(* Logix 5000 project; controller test vendor 1 type 14 code 106 rev 30.11; software revision 30.00 *)

TASK MainTask (continuous, watchdog 500 ms) : MainProgram

MODULES
   Local : vendor 1 type 14 code 106 (Compact 0, rev 30.11)
END_MODULES

TYPE DateTime :   // Date and TimeOfDay (absolute) or Time (duration/interval)
STRUCT
   Yr : DINT;   // Year(s)
   Mo : DINT;   // Month(s)
   Da : DINT;   // Day(s)
   Hr : DINT;   // Hour(s)
   Min : DINT;   // Minute(s)
   Sec : DINT;   // Second(s)
   uSec : DINT;   // Microsecond(s)
END_STRUCT
END_TYPE

TYPE Diesel_User :
STRUCT
   user_number : DINT;   // user number/any 32 bit interger
   gallons_in : REAL;   // user gallons filled
   gallons_out : REAL;   // user gallons dispenced
   last_Tx : DateTime;   // date and time of last transaction
END_STRUCT
END_TYPE

ADD_ON_INSTRUCTION CALC_HORZ_TANK   (* revision 1.0, vendor truvision *)
// Gallons in a Horizontal Tank
// Help:
// Add on instruction to calculate the gallons in a cylindrical horizontal tank, based on the diameter of the tank, the length of the tank, and the distance from the surface of the liquid to the top of the tank.
VAR_INPUT
   cyl_dia : REAL; {required}
   cyl_len : REAL; {required}
   dist : REAL; {required}
END_VAR
VAR_IN_OUT
   gal : REAL; {required}
END_VAR
VAR
   al : REAL; {access None}
   vol : REAL; {access None}
   cyl_rad : REAL; {access None}
END_VAR

ROUTINE Logic   (* structured text *)
   cyl_rad:=cyl_dia/2;
   al:=3.1415*cyl_rad**2-cyl_rad**2*ACOS((cyl_rad-dist)/cyl_rad)+(cyl_rad-dist)*SQRT(2*cyl_rad*dist-dist**2);
   vol:=al*cyl_len;
   gal:=vol*7.48052;
END_ROUTINE
END_ADD_ON_INSTRUCTION

VAR_GLOBAL   (* controller tags *)
   al : REAL := 39.230095;   // tank end cap area output
   always_off : BOOL;
   Check_Diesel_User : CONTROL := (LEN := 50);
   Current_Diesel_User : Diesel_User;
   cyl_h : REAL := 5.0;   // distance from the top of tank to the liquid
   cyl_rad : REAL := 5.0;   // tank drum radius
   Data_Enter_PB : BOOL;
   Date_Time : DateTime;
   Diesel_User_Gallons : REAL;
   Diesel_User_Number : DINT;
   Diesel_Users : Diesel_User[50] := ([0].user_number := 100, [1].user_number := 200, [2].user_number := 300, [3].user_number := 400, [4].user_number := 500);
   found : BOOL;
   gal : REAL := 2934.6152;   // volume output in gallons
   hi : REAL := 5.0;
   le : REAL := 10.0;
   length : REAL := 10.0;   // length of tank
   OffRoad_PB : BOOL;
   OffRoad_Selected : BOOL;
   OnRoad_PB : BOOL;
   OnRoad_Selected : BOOL;
   pi : REAL := 3.14;   // constant pi
   ra : REAL := 10.0;
   Reset_Diesel_Pump : BOOL;
   stuff : BOOL := 1;
   tk : CALC_HORZ_TANK;
   tk1 : CALC_HORZ_TANK := (cyl_dia := 10.0, cyl_len := 10.0, dist := 5.0);
   tk1_gallons : REAL := 2937.4194;
   vol : REAL := 392.30096;   // volume output in cubic feet
END_VAR

PROGRAM MainProgram   (* main routine MainRoutine *)

ROUTINE MainRoutine   (* ladder *)
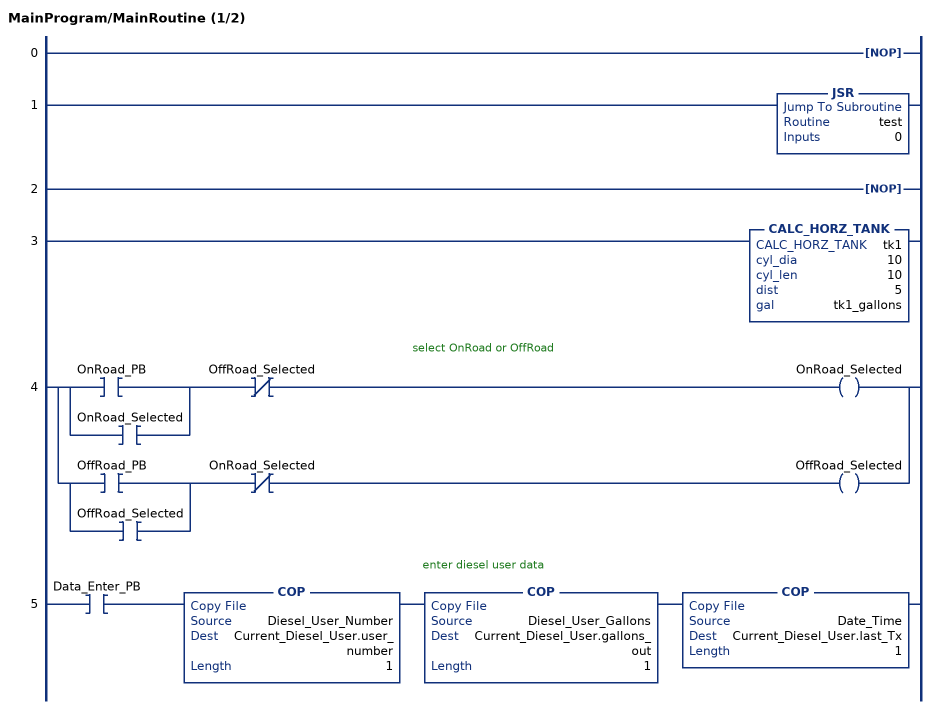
   0: NOP();
   1: JSR(test,0);
   2: NOP();
   3: CALC_HORZ_TANK(tk1,10,10,5,tk1_gallons);
   // select OnRoad or OffRoad
   4: [[XIC(OnRoad_PB) ,XIC(OnRoad_Selected) ] XIO(OffRoad_Selected) OTE(OnRoad_Selected) ,[XIC(OffRoad_PB) ,XIC(OffRoad_Selected) ] XIO(OnRoad_Selected) OTE(OffRoad_Selected) ];
   // enter diesel user data
   5: XIC(Data_Enter_PB)COP(Diesel_User_Number,Current_Diesel_User.user_number,1)COP(Diesel_User_Gallons,Current_Diesel_User.gallons_out,1)COP(Date_Time,Current_Diesel_User.last_Tx,1);
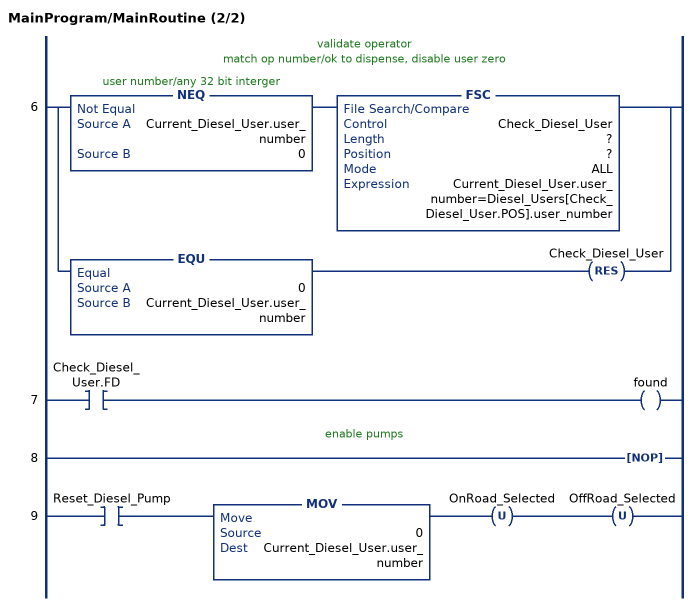
   // validate operator
   // match op number/ok to dispense, disable user zero
   6: [NEQ(Current_Diesel_User.user_number,0) FSC(Check_Diesel_User,?,?,ALL,Current_Diesel_User.user_number=Diesel_Users[Check_Diesel_User.POS].user_number) ,EQU(0,Current_Diesel_User.user_number) RES(Check_Diesel_User) ];
   7: XIC(Check_Diesel_User.FD)OTE(found);
   // enable pumps
   8: NOP();
   9: XIC(Reset_Diesel_Pump)MOV(0,Current_Diesel_User.user_number)OTU(OnRoad_Selected)OTU(OffRoad_Selected);
END_ROUTINE

ROUTINE test   (* structured text *)
   
   al:=pi*cyl_rad**2-cyl_rad**2*ACOS((cyl_rad-cyl_h)/cyl_rad)+(cyl_rad-cyl_h)*SQRT(2*cyl_rad*cyl_h-cyl_h**2);
   vol:=al*length;
   gal:=vol*7.48052;
   
   
   
END_ROUTINE
END_PROGRAM
